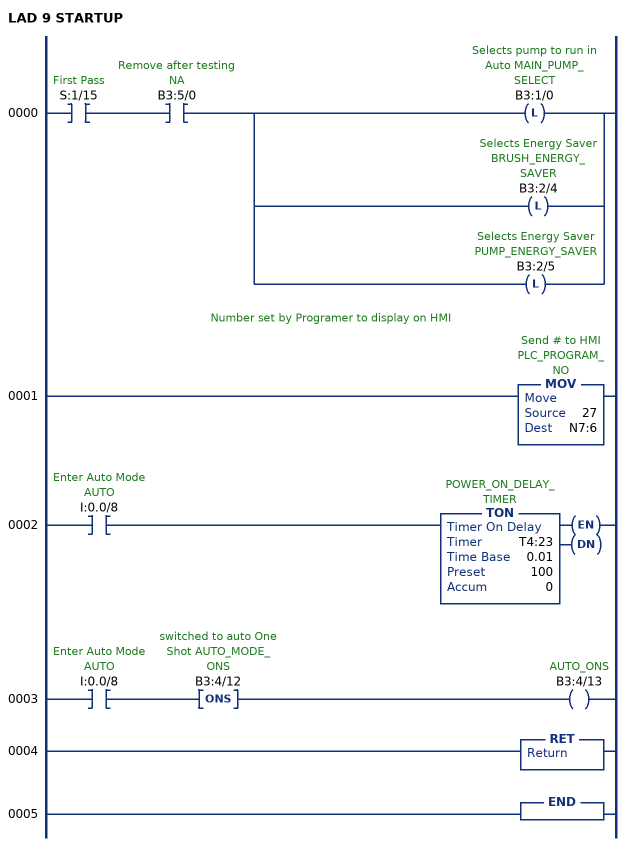
% Rung: 0 %
SOR XIC S:1/15 XIC B3:5/0 BST OTL B3:1/0 NXB BST OTL B3:2/4 NXB OTL B3:2/5 BND BND EOR
%   S:1/15  "First Pass" %
%   B3:5/0  NA  "Remove after testing" %
%   B3:1/0  MAIN_PUMP_SELECT  "Selects pump to run in Auto" %
%   B3:2/4  BRUSH_ENERGY_SAVER  "Selects Energy Saver" %
%   B3:2/5  PUMP_ENERGY_SAVER  "Selects Energy Saver" %
% Rung: 1 %
% Number set by Programer to display on HMI %
SOR MOV 27 N7:6 EOR
%   N7:6  PLC_PROGRAM_NO  "Send # to HMI" %
% Rung: 2 %
SOR XIC I:0.0/8 TON T4:23 0.01 100 0 EOR
%   I:0.0/8  AUTO  "Enter Auto Mode" %
%   T4:23  POWER_ON_DELAY_TIMER %
% Rung: 3 %
SOR XIC I:0.0/8 ONS B3:4/12 OTE B3:4/13 EOR
%   I:0.0/8  AUTO  "Enter Auto Mode" %
%   B3:4/12  AUTO_MODE_ONS  "switched to auto One Shot" %
%   B3:4/13  AUTO_ONS %
% Rung: 4 %
SOR RET EOR
% Rung: 5 %
SOR END EOR

LADDER 10 "FAULTS"    % Faults %
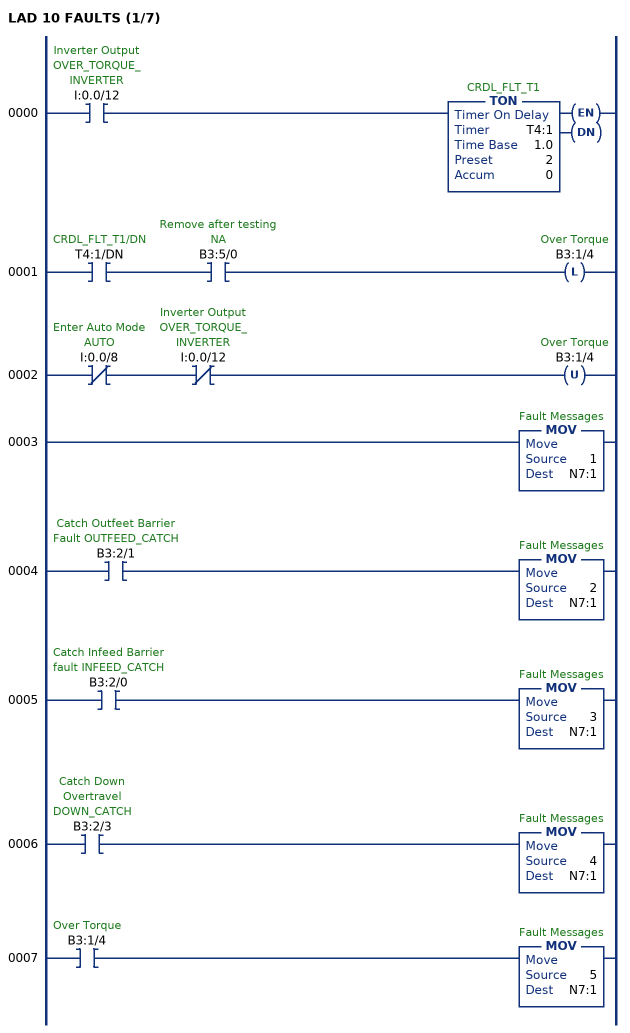
% Rung: 0 %
SOR XIC I:0.0/12 TON T4:1 1.0 2 0 EOR
%   I:0.0/12  OVER_TORQUE_INVERTER  "Inverter Output" %
%   T4:1  CRDL_FLT_T1 %
% Rung: 1 %
SOR XIC T4:1/DN XIC B3:5/0 OTL B3:1/4 EOR
%   T4:1  CRDL_FLT_T1 %
%   B3:5/0  NA  "Remove after testing" %
%   B3:1/4  "Over Torque" %
% Rung: 2 %
SOR XIO I:0.0/8 XIO I:0.0/12 OTU B3:1/4 EOR
%   I:0.0/8  AUTO  "Enter Auto Mode" %
%   I:0.0/12  OVER_TORQUE_INVERTER  "Inverter Output" %
%   B3:1/4  "Over Torque" %
% Rung: 3 %
SOR MOV 1 N7:1 EOR
%   N7:1  "Fault Messages" %
% Rung: 4 %
SOR XIC B3:2/1 MOV 2 N7:1 EOR
%   B3:2/1  OUTFEED_CATCH  "Catch Outfeet Barrier Fault" %
%   N7:1  "Fault Messages" %
% Rung: 5 %
SOR XIC B3:2/0 MOV 3 N7:1 EOR
%   B3:2/0  INFEED_CATCH  "Catch Infeed Barrier fault" %
%   N7:1  "Fault Messages" %
% Rung: 6 %
SOR XIC B3:2/3 MOV 4 N7:1 EOR
%   B3:2/3  DOWN_CATCH  "Catch Down Overtravel" %
%   N7:1  "Fault Messages" %
% Rung: 7 %
SOR XIC B3:1/4 MOV 5 N7:1 EOR
%   B3:1/4  "Over Torque" %
%   N7:1  "Fault Messages" %

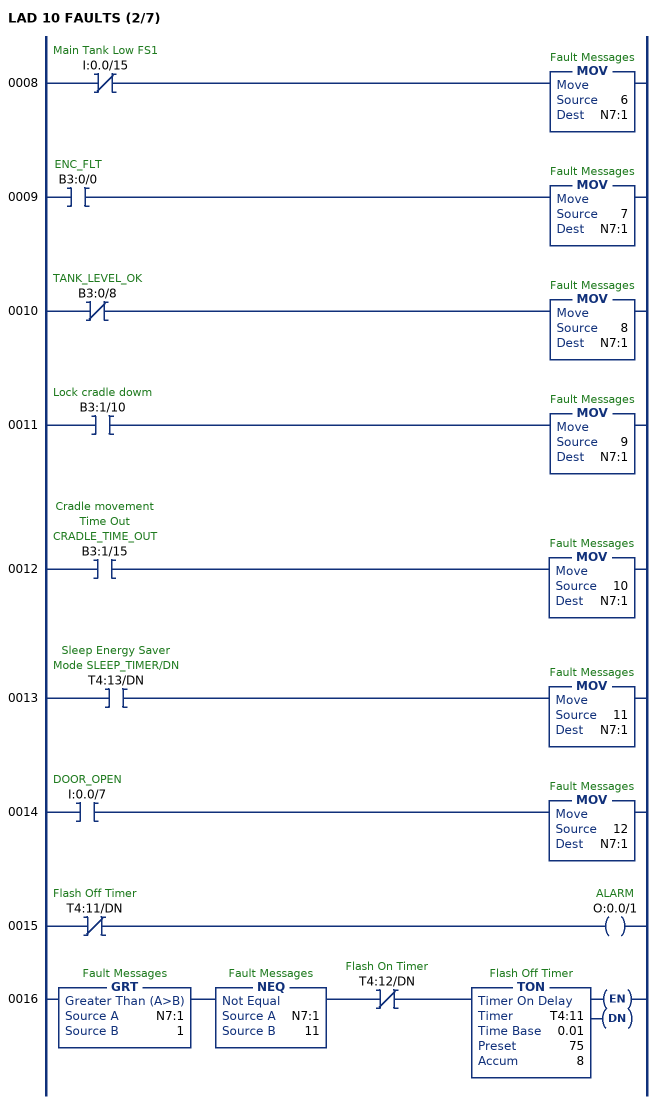
% Rung: 8 %
SOR XIO I:0.0/15 MOV 6 N7:1 EOR
%   I:0.0/15  FS1  "Main Tank Low" %
%   N7:1  "Fault Messages" %
% Rung: 9 %
SOR XIC B3:0/0 MOV 7 N7:1 EOR
%   B3:0/0  ENC_FLT %
%   N7:1  "Fault Messages" %
% Rung: 10 %
SOR XIO B3:0/8 MOV 8 N7:1 EOR
%   B3:0/8  TANK_LEVEL_OK %
%   N7:1  "Fault Messages" %
% Rung: 11 %
SOR XIC B3:1/10 MOV 9 N7:1 EOR
%   B3:1/10  "Lock cradle dowm" %
%   N7:1  "Fault Messages" %
% Rung: 12 %
SOR XIC B3:1/15 MOV 10 N7:1 EOR
%   B3:1/15  CRADLE_TIME_OUT  "Cradle movement Time Out" %
%   N7:1  "Fault Messages" %
% Rung: 13 %
SOR XIC T4:13/DN MOV 11 N7:1 EOR
%   T4:13  SLEEP_TIMER  "Sleep Energy Saver Mode" %
%   N7:1  "Fault Messages" %
% Rung: 14 %
SOR XIC I:0.0/7 MOV 12 N7:1 EOR
%   I:0.0/7  DOOR_OPEN %
%   N7:1  "Fault Messages" %
% Rung: 15 %
SOR XIO T4:11/DN OTE O:0.0/1 EOR
%   T4:11  "Flash Off Timer" %
%   O:0.0/1  ALARM %
% Rung: 16 %
SOR GRT N7:1 1 NEQ N7:1 11 XIO T4:12/DN TON T4:11 0.01 75 8 EOR
%   N7:1  "Fault Messages" %
%   T4:12  "Flash On Timer" %
%   T4:11  "Flash Off Timer" %

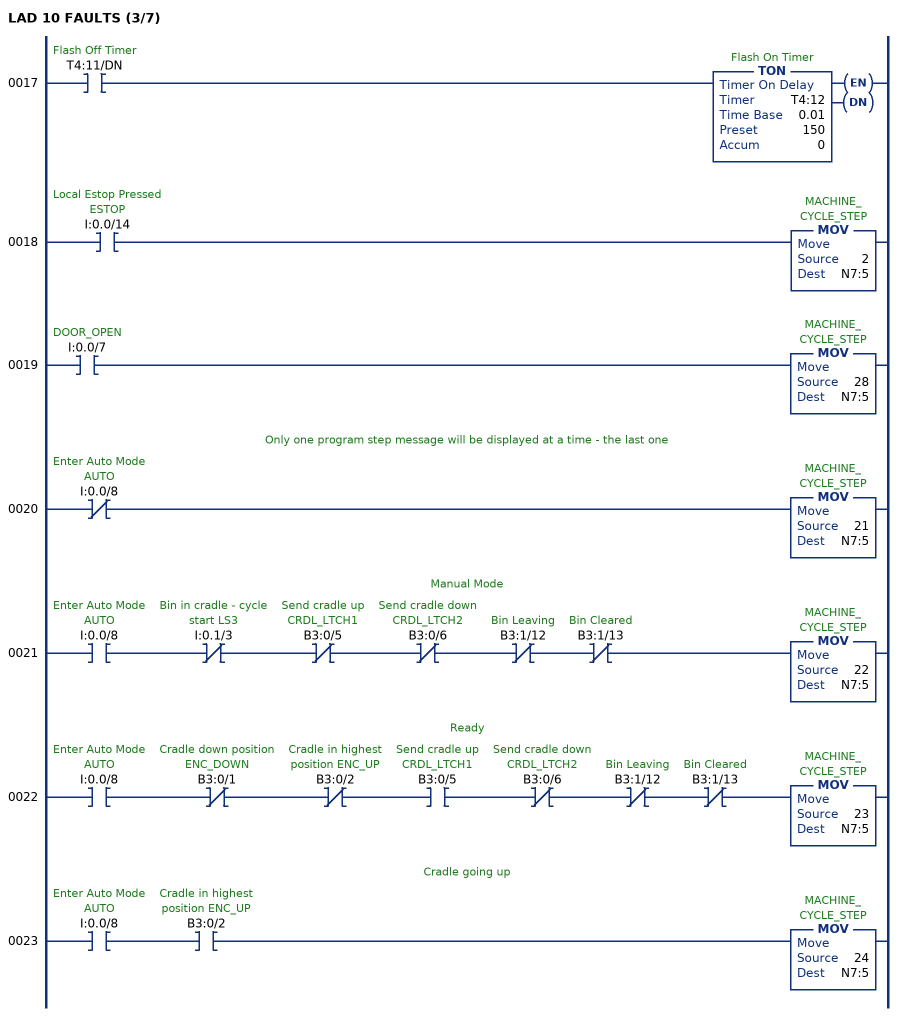
% Rung: 17 %
SOR XIC T4:11/DN TON T4:12 0.01 150 0 EOR
%   T4:11  "Flash Off Timer" %
%   T4:12  "Flash On Timer" %
% Rung: 18 %
SOR XIC I:0.0/14 MOV 2 N7:5 EOR
%   I:0.0/14  ESTOP  "Local Estop Pressed" %
%   N7:5  MACHINE_CYCLE_STEP %
% Rung: 19 %
SOR XIC I:0.0/7 MOV 28 N7:5 EOR
%   I:0.0/7  DOOR_OPEN %
%   N7:5  MACHINE_CYCLE_STEP %
% Rung: 20 %
% Only one program step message will be displayed at a time - the last one %
SOR XIO I:0.0/8 MOV 21 N7:5 EOR
%   I:0.0/8  AUTO  "Enter Auto Mode" %
%   N7:5  MACHINE_CYCLE_STEP %
% Rung: 21 %
% Manual Mode %
SOR XIC I:0.0/8 XIO I:0.1/3 XIO B3:0/5 XIO B3:0/6 XIO B3:1/12 XIO B3:1/13 MOV 22 N7:5 EOR
%   I:0.0/8  AUTO  "Enter Auto Mode" %
%   I:0.1/3  LS3  "Bin in cradle - cycle start" %
%   B3:0/5  CRDL_LTCH1  "Send cradle up" %
%   B3:0/6  CRDL_LTCH2  "Send cradle down" %
%   B3:1/12  "Bin Leaving" %
%   B3:1/13  "Bin Cleared" %
%   N7:5  MACHINE_CYCLE_STEP %
% Rung: 22 %
% Ready %
SOR XIC I:0.0/8 XIO B3:0/1 XIO B3:0/2 XIC B3:0/5 XIO B3:0/6 XIO B3:1/12 XIO B3:1/13 MOV 23 N7:5 EOR
%   I:0.0/8  AUTO  "Enter Auto Mode" %
%   B3:0/1  ENC_DOWN  "Cradle down position" %
%   B3:0/2  ENC_UP  "Cradle in highest position" %
%   B3:0/5  CRDL_LTCH1  "Send cradle up" %
%   B3:0/6  CRDL_LTCH2  "Send cradle down" %
%   B3:1/12  "Bin Leaving" %
%   B3:1/13  "Bin Cleared" %
%   N7:5  MACHINE_CYCLE_STEP %
% Rung: 23 %
% Cradle going up %
SOR XIC I:0.0/8 XIC B3:0/2 MOV 24 N7:5 EOR
%   I:0.0/8  AUTO  "Enter Auto Mode" %
%   B3:0/2  ENC_UP  "Cradle in highest position" %
%   N7:5  MACHINE_CYCLE_STEP %

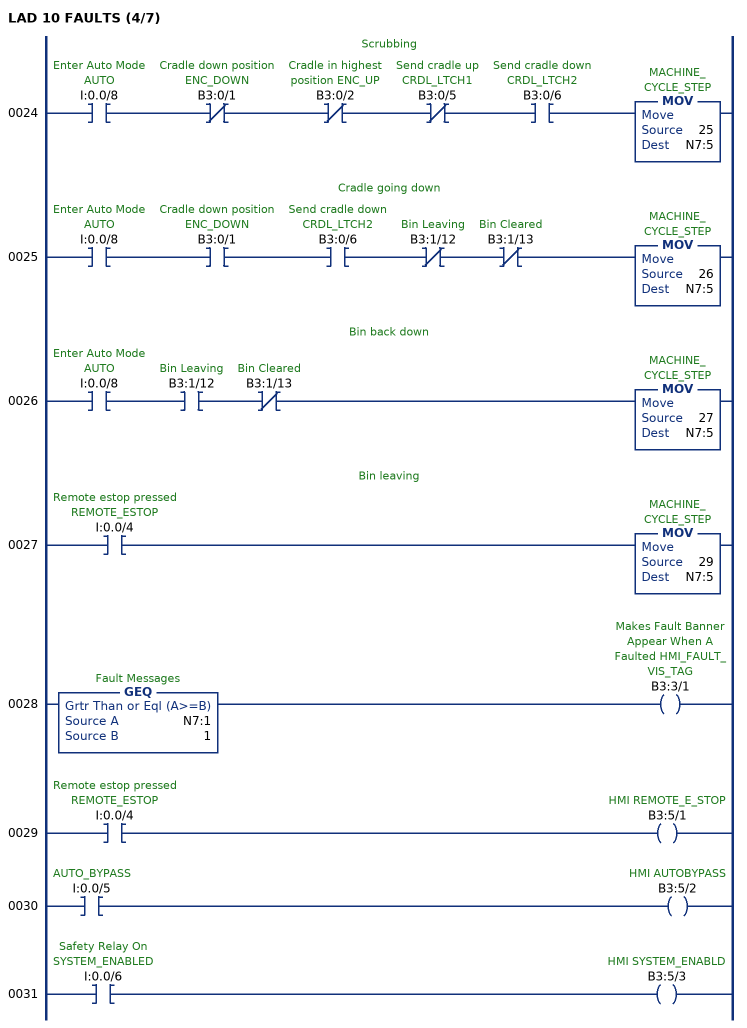
% Rung: 24 %
% Scrubbing %
SOR XIC I:0.0/8 XIO B3:0/1 XIO B3:0/2 XIO B3:0/5 XIC B3:0/6 MOV 25 N7:5 EOR
%   I:0.0/8  AUTO  "Enter Auto Mode" %
%   B3:0/1  ENC_DOWN  "Cradle down position" %
%   B3:0/2  ENC_UP  "Cradle in highest position" %
%   B3:0/5  CRDL_LTCH1  "Send cradle up" %
%   B3:0/6  CRDL_LTCH2  "Send cradle down" %
%   N7:5  MACHINE_CYCLE_STEP %
% Rung: 25 %
% Cradle going down %
SOR XIC I:0.0/8 XIC B3:0/1 XIC B3:0/6 XIO B3:1/12 XIO B3:1/13 MOV 26 N7:5 EOR
%   I:0.0/8  AUTO  "Enter Auto Mode" %
%   B3:0/1  ENC_DOWN  "Cradle down position" %
%   B3:0/6  CRDL_LTCH2  "Send cradle down" %
%   B3:1/12  "Bin Leaving" %
%   B3:1/13  "Bin Cleared" %
%   N7:5  MACHINE_CYCLE_STEP %
% Rung: 26 %
% Bin back down %
SOR XIC I:0.0/8 XIC B3:1/12 XIO B3:1/13 MOV 27 N7:5 EOR
%   I:0.0/8  AUTO  "Enter Auto Mode" %
%   B3:1/12  "Bin Leaving" %
%   B3:1/13  "Bin Cleared" %
%   N7:5  MACHINE_CYCLE_STEP %
% Rung: 27 %
% Bin leaving %
SOR XIC I:0.0/4 MOV 29 N7:5 EOR
%   I:0.0/4  REMOTE_ESTOP  "Remote estop pressed" %
%   N7:5  MACHINE_CYCLE_STEP %
% Rung: 28 %
SOR GEQ N7:1 1 OTE B3:3/1 EOR
%   N7:1  "Fault Messages" %
%   B3:3/1  HMI_FAULT_VIS_TAG  "Makes Fault Banner Appear When A Faulted" %
% Rung: 29 %
SOR XIC I:0.0/4 OTE B3:5/1 EOR
%   I:0.0/4  REMOTE_ESTOP  "Remote estop pressed" %
%   B3:5/1  REMOTE_E_STOP  "HMI" %
% Rung: 30 %
SOR XIC I:0.0/5 OTE B3:5/2 EOR
%   I:0.0/5  AUTO_BYPASS %
%   B3:5/2  AUTOBYPASS  "HMI" %
% Rung: 31 %
SOR XIC I:0.0/6 OTE B3:5/3 EOR
%   I:0.0/6  SYSTEM_ENABLED  "Safety Relay On" %
%   B3:5/3  SYSTEM_ENABLD  "HMI" %

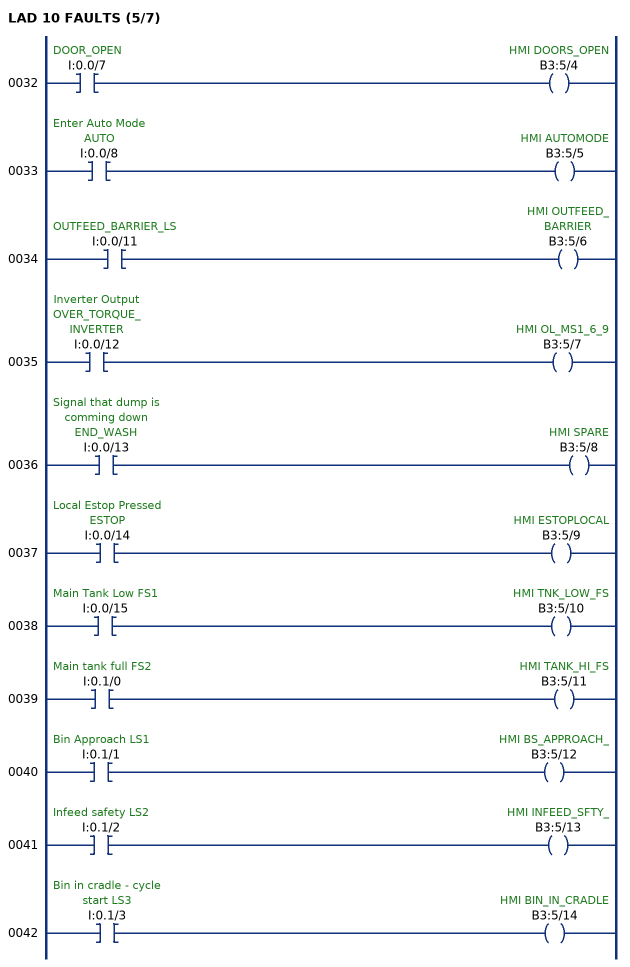
% Rung: 32 %
SOR XIC I:0.0/7 OTE B3:5/4 EOR
%   I:0.0/7  DOOR_OPEN %
%   B3:5/4  DOORS_OPEN  "HMI" %
% Rung: 33 %
SOR XIC I:0.0/8 OTE B3:5/5 EOR
%   I:0.0/8  AUTO  "Enter Auto Mode" %
%   B3:5/5  AUTOMODE  "HMI" %
% Rung: 34 %
SOR XIC I:0.0/11 OTE B3:5/6 EOR
%   I:0.0/11  OUTFEED_BARRIER_LS %
%   B3:5/6  OUTFEED_BARRIER  "HMI" %
% Rung: 35 %
SOR XIC I:0.0/12 OTE B3:5/7 EOR
%   I:0.0/12  OVER_TORQUE_INVERTER  "Inverter Output" %
%   B3:5/7  OL_MS1_6_9  "HMI" %
% Rung: 36 %
SOR XIC I:0.0/13 OTE B3:5/8 EOR
%   I:0.0/13  END_WASH  "Signal that dump is comming down" %
%   B3:5/8  SPARE  "HMI" %
% Rung: 37 %
SOR XIC I:0.0/14 OTE B3:5/9 EOR
%   I:0.0/14  ESTOP  "Local Estop Pressed" %
%   B3:5/9  ESTOPLOCAL  "HMI" %
% Rung: 38 %
SOR XIC I:0.0/15 OTE B3:5/10 EOR
%   I:0.0/15  FS1  "Main Tank Low" %
%   B3:5/10  TNK_LOW_FS  "HMI" %
% Rung: 39 %
SOR XIC I:0.1/0 OTE B3:5/11 EOR
%   I:0.1/0  FS2  "Main tank full" %
%   B3:5/11  TANK_HI_FS  "HMI" %
% Rung: 40 %
SOR XIC I:0.1/1 OTE B3:5/12 EOR
%   I:0.1/1  LS1  "Bin Approach" %
%   B3:5/12  BS_APPROACH_  "HMI" %
% Rung: 41 %
SOR XIC I:0.1/2 OTE B3:5/13 EOR
%   I:0.1/2  LS2  "Infeed safety" %
%   B3:5/13  INFEED_SFTY_  "HMI" %
% Rung: 42 %
SOR XIC I:0.1/3 OTE B3:5/14 EOR
%   I:0.1/3  LS3  "Bin in cradle - cycle start" %
%   B3:5/14  BIN_IN_CRADLE  "HMI" %

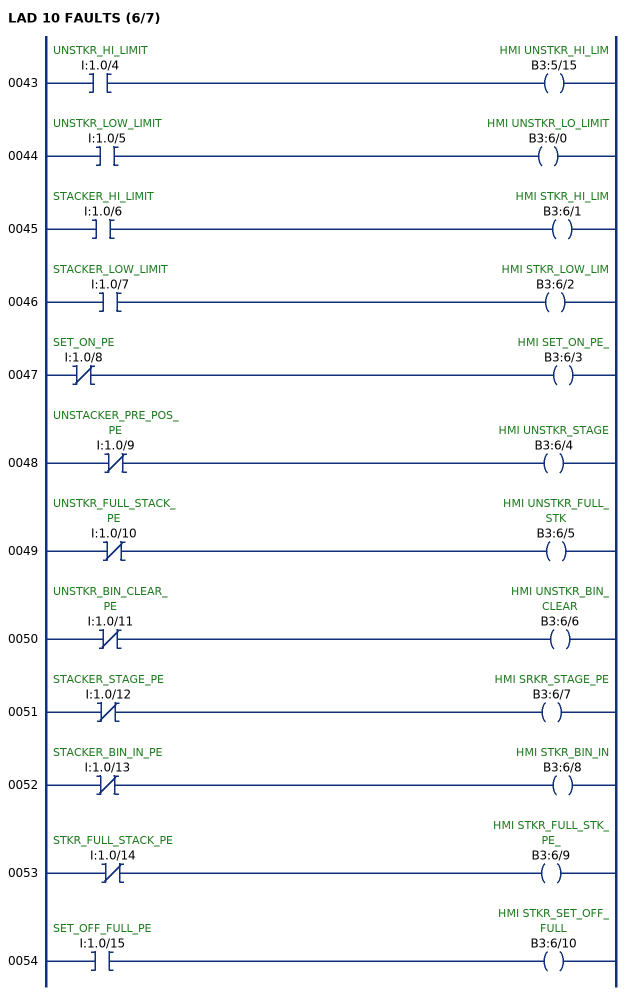
% Rung: 43 %
SOR XIC I:1.0/4 OTE B3:5/15 EOR
%   I:1.0/4  UNSTKR_HI_LIMIT %
%   B3:5/15  UNSTKR_HI_LIM  "HMI" %
% Rung: 44 %
SOR XIC I:1.0/5 OTE B3:6/0 EOR
%   I:1.0/5  UNSTKR_LOW_LIMIT %
%   B3:6/0  UNSTKR_LO_LIMIT  "HMI" %
% Rung: 45 %
SOR XIC I:1.0/6 OTE B3:6/1 EOR
%   I:1.0/6  STACKER_HI_LIMIT %
%   B3:6/1  STKR_HI_LIM  "HMI" %
% Rung: 46 %
SOR XIC I:1.0/7 OTE B3:6/2 EOR
%   I:1.0/7  STACKER_LOW_LIMIT %
%   B3:6/2  STKR_LOW_LIM  "HMI" %
% Rung: 47 %
SOR XIO I:1.0/8 OTE B3:6/3 EOR
%   I:1.0/8  SET_ON_PE %
%   B3:6/3  SET_ON_PE_  "HMI" %
% Rung: 48 %
SOR XIO I:1.0/9 OTE B3:6/4 EOR
%   I:1.0/9  UNSTACKER_PRE_POS_PE %
%   B3:6/4  UNSTKR_STAGE  "HMI" %
% Rung: 49 %
SOR XIO I:1.0/10 OTE B3:6/5 EOR
%   I:1.0/10  UNSTKR_FULL_STACK_PE %
%   B3:6/5  UNSTKR_FULL_STK  "HMI" %
% Rung: 50 %
SOR XIO I:1.0/11 OTE B3:6/6 EOR
%   I:1.0/11  UNSTKR_BIN_CLEAR_PE %
%   B3:6/6  UNSTKR_BIN_CLEAR  "HMI" %
% Rung: 51 %
SOR XIO I:1.0/12 OTE B3:6/7 EOR
%   I:1.0/12  STACKER_STAGE_PE %
%   B3:6/7  SRKR_STAGE_PE  "HMI" %
% Rung: 52 %
SOR XIO I:1.0/13 OTE B3:6/8 EOR
%   I:1.0/13  STACKER_BIN_IN_PE %
%   B3:6/8  STKR_BIN_IN  "HMI" %
% Rung: 53 %
SOR XIO I:1.0/14 OTE B3:6/9 EOR
%   I:1.0/14  STKR_FULL_STACK_PE %
%   B3:6/9  STKR_FULL_STK_PE_  "HMI" %
% Rung: 54 %
SOR XIC I:1.0/15 OTE B3:6/10 EOR
%   I:1.0/15  SET_OFF_FULL_PE %
%   B3:6/10  STKR_SET_OFF_FULL  "HMI" %

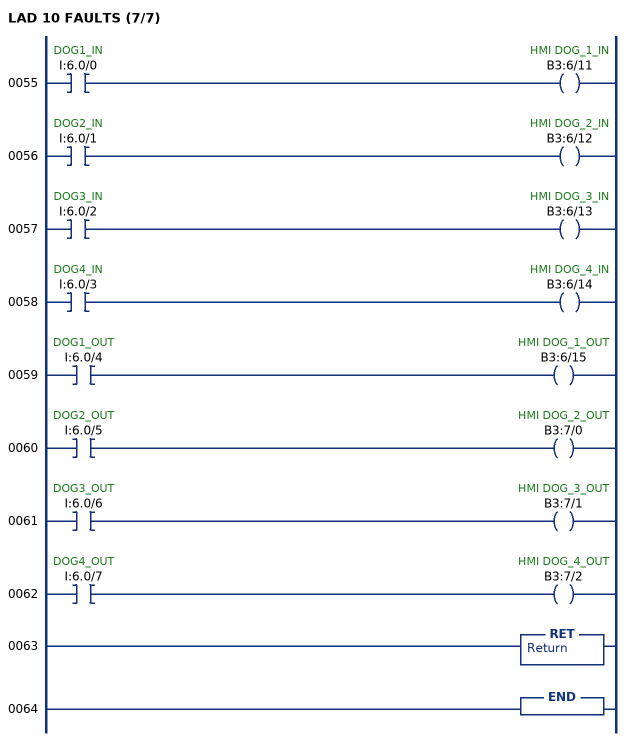
% Rung: 55 %
SOR XIC I:6.0/0 OTE B3:6/11 EOR
%   I:6.0/0  DOG1_IN %
%   B3:6/11  DOG_1_IN  "HMI" %
% Rung: 56 %
SOR XIC I:6.0/1 OTE B3:6/12 EOR
%   I:6.0/1  DOG2_IN %
%   B3:6/12  DOG_2_IN  "HMI" %
% Rung: 57 %
SOR XIC I:6.0/2 OTE B3:6/13 EOR
%   I:6.0/2  DOG3_IN %
%   B3:6/13  DOG_3_IN  "HMI" %
% Rung: 58 %
SOR XIC I:6.0/3 OTE B3:6/14 EOR
%   I:6.0/3  DOG4_IN %
%   B3:6/14  DOG_4_IN  "HMI" %
% Rung: 59 %
SOR XIC I:6.0/4 OTE B3:6/15 EOR
%   I:6.0/4  DOG1_OUT %
%   B3:6/15  DOG_1_OUT  "HMI" %
% Rung: 60 %
SOR XIC I:6.0/5 OTE B3:7/0 EOR
%   I:6.0/5  DOG2_OUT %
%   B3:7/0  DOG_2_OUT  "HMI" %
% Rung: 61 %
SOR XIC I:6.0/6 OTE B3:7/1 EOR
%   I:6.0/6  DOG3_OUT %
%   B3:7/1  DOG_3_OUT  "HMI" %
% Rung: 62 %
SOR XIC I:6.0/7 OTE B3:7/2 EOR
%   I:6.0/7  DOG4_OUT %
%   B3:7/2  DOG_4_OUT  "HMI" %
% Rung: 63 %
SOR RET EOR
% Rung: 64 %
SOR END EOR

LADDER 11 "HSC"    % Bin Scrubber Cradle %
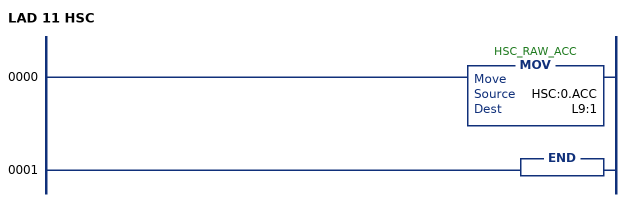
% Rung: 0 %
SOR MOV HSC:0.ACC L9:1 EOR
%   L9:1  HSC_RAW_ACC %
% Rung: 1 %
SOR END EOR

OTHER DOCUMENTED ADDRESSES
  I:0.0/0  ENCODER_HSC  "Pink"
  I:0.0/1  ENCODER_HSC_  "Yellow"
  I:0.0/2  NOT_USED
  I:0.0/3  NOT_USED_
  I:1.0/0  BS_CRADLE_OL
  I:1.0/1  BS_BRUSH_OL
  I:1.0/2  UNSTACKER_CRADLE_OL
  I:1.0/3  STACKER_CRADLE_OL
  I:5.0/12  DOGS_IN_LS
  I:5.0/13  DOGS_OUT_LS
  I:5.0/14  SPARE__
  I:5.0/15  SPARE___
  O:0.0/7  NOT_USED__
  O:2.0/4  SANITARY_PUMP
  O:2.0/7  EXTRA__
  O:3.0/3  NOT_USED___
  O:3.0/7  NOT_USED____

DATA TABLE (non-zero values as saved)
DATA B3
% B3:0 % 0X5112 0X0001 0X4850 0X0602 0X8044 0X2C58 0X8080 0X0477 0X0000
DATA T4
% .PRE .ACC %
% T4:0 % 100 100
% T4:1 % 2 0
% T4:2 % 3 3
% T4:3 % 1000 0
% T4:4 % 10 10
% T4:5 % 30 30
% T4:6 % 1 1
% T4:7 % 30 30
% T4:8 % 30 0
% T4:9 % 2 0
% T4:10 % 1 1
% T4:11 % 75 8
% T4:12 % 150 0
% T4:13 % 180 0
% T4:14 % 1 0
% T4:15 % 10 0
% T4:16 % 10 0
% T4:17 % 1 0
% T4:18 % 100 0
% T4:19 % 10 10
% T4:20 % 50 0
% T4:21 % 100 0
% T4:22 % 100 0
% T4:23 % 100 0
% T4:24 % 500 500
% T4:25 % 6 0
% T4:27 % 10 0
% T4:28 % 25 0
% T4:29 % 2 0
% T4:30 % 7 7
% T4:31 % 1 0
% T4:32 % 6100 6100
% T4:33 % 2 2
DATA N7
% N7:0 % 16839 12 12 60 59 21 27 10175 4 16186
% N7:10 % 12491 0 88 77 2 98 0 10 77 115
% N7:20 % 15
DATA F8
% F8:0 % 16138
DATA L9
% L9:0 % 0 1443 3
